Fanuc KAREL source: kt00291.KL

-- PROVISIONAL review KL for V940-1; original PC SHA256 740538cfa0a13b65d434d8f439b6a6e9aafdf97abf64a734e6ffddd7cb0017a3
-- Incomplete behavior may be omitted. Consult companion uncertainty JSON. Do not deploy.
PROGRAM KT00291
%NOLOCKGROUP
VAR
  OUT : BOOLEAN
-- UNRESOLVED_DECL V1 type=000013
-- UNRESOLVED_DECL V2 type=000013
BEGIN
  -- V9_ZERO_TABLE_METADATA_HINT layout=0001; no indexed target words; source/name/runtime held
  -- UNRESOLVED_PC offsets 5-20; opcodes 2E,22,32,35
  -- UNRESOLVED_PC offsets 25-40; opcodes 2E,22,32,35
  -- UNRESOLVED_PC offsets 45-60; opcodes 2E,22,32,35
  -- UNRESOLVED_PC offsets 65-80; opcodes 2E,22,32,35
  -- UNRESOLVED_PC offsets 85-108; opcodes 49,49,95,23
  -- UNRESOLVED_PC offsets 113-117; opcodes 7F
END KT00291
